FUNCTION_BLOCK OpticalSensor IMPLEMENTS ITF_BinarySensor
VAR_INPUT
END_VAR
VAR_OUTPUT
END_VAR
VAR
	//Hardware
	//{attribute 'OPC.UA.DA' := '1'}
	DI_WPLight AT %I* : BOOL;
END_VAR

PROPERTY Value : BOOL
GET
Value := DI_WPLight;
END_GET
END_PROPERTY

END_FUNCTION_BLOCK

(* stored: Version 1.1.0.1, ProductVersion 3.1.4024.9
   POU OpticalSensor: Id {cd0e5918-4a05-4022-bff4-d1699e9fcf32}, SpecialFunc None
   Property Value: Id {9e1f82ad-8a05-407c-b8b1-d65027c57492}
   Get Get: Id {8ba229cf-4496-4d8f-ba57-2c9175f53097} *)
